// TIA Portal project "Bottle_line" (V15.1)

(* hardware
DEVICE "S7-1200 station_1"  S7-1200 Station
   slot 0: "Rack_0"  S7-1200 Rack  Rack  V1.0
   slot 1: "PLC_1"  CPU 1214C AC/DC/Rly  6ES7 214-1BG40-0XB0  V4.2
*)

// ===== PLC "PLC_1"  CPU 1214C AC/DC/Rly =====

VAR_GLOBAL   // PLC tag table "Default tag table"
   "System_Byte" AT %MB1 : Byte;
   "FirstScan" AT %M1.0 : Bool;
   "DiagStatusUpdate" AT %M1.1 : Bool;
   "AlwaysTRUE" AT %M1.2 : Bool;
   "AlwaysFALSE" AT %M1.3 : Bool;
   "Clock_Byte" AT %MB0 : Byte;
   "Clock_10Hz" AT %M0.0 : Bool;
   "Clock_5Hz" AT %M0.1 : Bool;
   "Clock_2.5Hz" AT %M0.2 : Bool;
   "Clock_2Hz" AT %M0.3 : Bool;
   "Clock_1.25Hz" AT %M0.4 : Bool;
   "Clock_1Hz" AT %M0.5 : Bool;
   "Clock_0.625Hz" AT %M0.6 : Bool;
   "Clock_0.5Hz" AT %M0.7 : Bool;
   "System_Byte(1)" AT %MB1 : Byte;
END_VAR

VAR_GLOBAL   // PLC tag table "Tag table_1"
   "LevelSensor" AT %IW56 : Word;
   "FlowMeter" AT %IW58 : Word;
   "FillTankValve" AT %QW56 : Word;
   "DrainValve" AT %QW58 : Word;
   "Start" AT %I20.0 : Bool;
   "Stop" AT %I20.1 : Bool;
   "Pause" AT %I20.2 : Bool;
   "BottleDetector" AT %I20.3 : Bool;
   "BottleCounter" AT %I20.4 : Bool;
   "BottleDetect" AT %I20.5 : Bool;
   "Emitter" AT %Q20.0 : Bool;
   "Conveyor1" AT %Q20.1 : Bool;
   "Conveyor2" AT %Q20.2 : Bool;
   "Conveyor3" AT %Q20.3 : Bool;
   "Conveyor4" AT %Q20.4 : Bool;
   "Conveyor5" AT %Q20.5 : Bool;
   "RollerStop" AT %Q20.6 : Bool;
   "RoboticArmZ" AT %Q20.7 : Bool;
   "GrabArmZ" AT %Q21.0 : Bool;
   "FillingLED" AT %Q21.1 : Bool;
   "GreenLED" AT %Q21.2 : Bool;
   "RedLEd" AT %Q21.3 : Bool;
   "YellowLED" AT %Q21.4 : Bool;
   "CounterDisplay" AT %QW60 : Word;
END_VAR

DATA_BLOCK "Bottle_Filling_DB"   // DB1
{ S7_Optimized_Access := 'TRUE' }
VERSION : 0.1
// stored: InstanceOfName Bottle_Filling
"Bottle_Filling"
BEGIN
END_DATA_BLOCK

DATA_BLOCK "Data"   // DB3
{ S7_Optimized_Access := 'TRUE' }
VERSION : 0.1
   VAR
      "SPTank(mm)" : Int := 3000;
      "PVTank(mm)" : Real;
      EnablePID : Bool;
      Norm : Real;
      "Caudal(m3/s)" : Real;
      bottleReset : Bool;
      "PVBottle(L)" : Real;
      "SPBottle(L)" : Real;
      BottleFill : Bool;
   END_VAR
BEGIN
END_DATA_BLOCK

DATA_BLOCK "Integration_DB"   // DB4
{ S7_Optimized_Access := 'TRUE' }
VERSION : 0.1
// stored: InstanceOfName Integration
"Integration"
BEGIN
END_DATA_BLOCK

DATA_BLOCK "TON_DB"   // DB7
{ S7_Optimized_Access := 'TRUE' }
VERSION : 0.1
// stored: InstanceOfName TON
"TON"
BEGIN
END_DATA_BLOCK

// folder: System blocks/Program resources

DATA_BLOCK "IEC_Timer_0_DB"   // DB6
{ S7_Optimized_Access := 'TRUE' }
AUTHOR : Simatic
FAMILY : IEC
NAME : IEC_TMR
VERSION : 1.0
// stored: InstanceOfName IEC_TIMER
"IEC_TIMER"
BEGIN
END_DATA_BLOCK

// folder: (top level)

FUNCTION_BLOCK "Bottle_Filling"   // FB1, LAD
{ S7_Optimized_Access := 'TRUE' }
VERSION : 0.1
   VAR_INPUT
      Start : Bool;
      Stop : Bool;
      Pause : Bool;
      BottleDetect : Bool;
      BottleCounter : Bool;
      BottleDetecter : Bool;
      LevelSensor : Int;
      "PV Bottle" : Real;
      "SP Bottle" : Real;
   END_VAR
   VAR_OUTPUT
      Emitter : Bool;
      Conveyor1 : Bool;
      Conveyor2 : Bool;
      Conveyor3 : Bool;
      Conveyor4 : Bool;
      Conveyor5 : Bool;
      RollerStop : Bool;
      RobotArmZ : Bool;
      GrabArmZ : Bool;
      FillingLED : Bool;
      GreenLED : Bool;
      RedLED : Bool;
      YellowLED : Bool;
      CounterDisplay : Int;
      LevelTank : Real;
      "BottleFilling X" : Bool;
      "BottleReset X" : Bool;
   END_VAR
   VAR
      K : Bool;
      Aux1 : Bool;
      Aux2 : Bool;
      X1_Emitter : Bool;
      X2_Emitter : Bool;
      Flanco1 : Bool;
      Flanco2 : Bool;
      Flanco3 : Bool;
      Flanco4 : Bool;
      XF : Bool;
      X1Stop : Bool;
      X2Stop : Bool;
      Detener : Bool;
      Norm : Real;
      "SP-error" : Real;
      "SP+error" : Real;
      "Counter" : CTU_INT;
      TON1 : "TON";
      TON3 : "TON";
      TON2 : "TON";
   END_VAR
   VAR_TEMP   // added for the SCL form of the ladder/FBD networks
      _w1 : Bool;
      _w2 : Bool;
   END_VAR
BEGIN

REGION Network 1
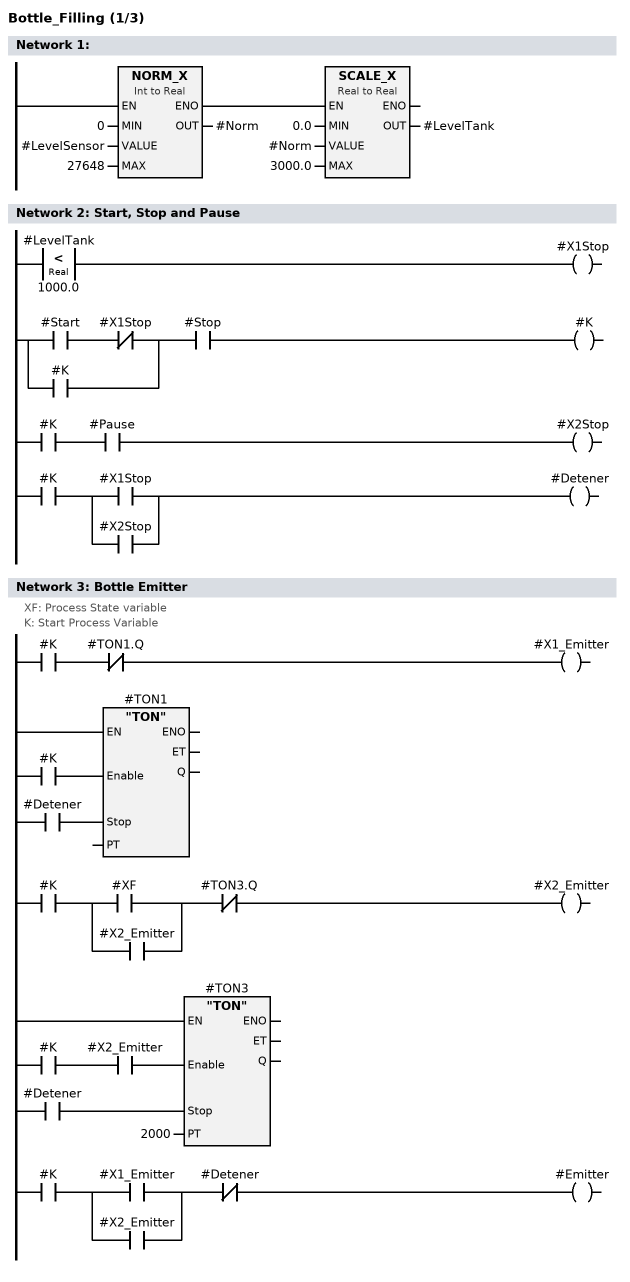
   RUNG wire#powerrail
      { S7_Templates := "[SrcType := Int, DestType := Real]" } Normalize(min := 0, value := #LevelSensor, max := 27648, out => #Norm)
      { S7_Templates := "[SrcType := Real, DestType := Real]" } Scale(min := 0.0, value := #Norm, max := 3000.0, out => #LevelTank)
   END_RUNG
   // the same network as SCL:
   #Norm := NORM_X(MIN := 0, VALUE := #LevelSensor, MAX := 27648);
   #LevelTank := SCALE_X(MIN := 0.0, VALUE := #Norm, MAX := 3000.0);
END_REGION

REGION Network 2: Start, Stop and Pause
   RUNG wire#powerrail
      { S7_Templates := "SrcType := Real" } LT_Contact(in1 := #LevelTank, in2 := 1000.0)
      Coil( #X1Stop )
   END_RUNG
   RUNG wire#powerrail
      Contact( #Start )
      I_Contact( #X1Stop )
      wire#w1
      Contact( #Stop )
      Coil( #K )
   END_RUNG
   RUNG wire#powerrail
      Contact( #K )
   END_RUNG wire#w1
   RUNG wire#powerrail
      Contact( #K )
      Contact( #Pause )
      Coil( #X2Stop )
   END_RUNG
   RUNG wire#powerrail
      Contact( #K )
      wire#w2
      Contact( #X1Stop )
      wire#w3
      Coil( #Detener )
   END_RUNG
   RUNG wire#w2
      Contact( #X2Stop )
   END_RUNG wire#w3
   // the same network as SCL:
   #X1Stop := #LevelTank < 1000.0;
   #K := ((#Start AND NOT #X1Stop) OR #K) AND #Stop;
   #X2Stop := #K AND #Pause;
   #Detener := #K AND (#X1Stop OR #X2Stop);
END_REGION

REGION Network 3: Bottle Emitter
   // XF: Process State variable
   // K: Start Process Variable
   RUNG wire#powerrail
      Contact( #K )
      I_Contact( #TON1.Q )
      Coil( #X1_Emitter )
   END_RUNG
   RUNG wire#powerrail
      #TON1(Enable := wire#w1, Stop := wire#w2, PT :=, ET =>, Q =>)
   END_RUNG
   RUNG wire#powerrail
      Contact( #K )
   END_RUNG wire#w1
   RUNG wire#powerrail
      Contact( #Detener )
   END_RUNG wire#w2
   RUNG wire#powerrail
      Contact( #K )
      wire#w3
      Contact( #XF )
      wire#w4
      I_Contact( #TON3.Q )
      Coil( #X2_Emitter )
   END_RUNG
   RUNG wire#w3
      Contact( #X2_Emitter )
   END_RUNG wire#w4
   RUNG wire#powerrail
      #TON3(Enable := wire#w5, Stop := wire#w6, PT := 2000, ET =>, Q =>)
   END_RUNG
   RUNG wire#powerrail
      Contact( #K )
      Contact( #X2_Emitter )
   END_RUNG wire#w5
   RUNG wire#powerrail
      Contact( #Detener )
   END_RUNG wire#w6
   RUNG wire#powerrail
      Contact( #K )
      wire#w7
      Contact( #X1_Emitter )
      wire#w8
      I_Contact( #Detener )
      Coil( #Emitter )
   END_RUNG
   RUNG wire#w7
      Contact( #X2_Emitter )
   END_RUNG wire#w8
   // the same network as SCL:
   #X1_Emitter := #K AND NOT #TON1.Q;
   #TON1(Enable := #K, Stop := #Detener);   // "TON"
   #X2_Emitter := #K AND (#XF OR #X2_Emitter) AND NOT #TON3.Q;
   #TON3(Enable := #K AND #X2_Emitter, Stop := #Detener, PT := 2000);   // "TON"
   #Emitter := #K AND (#X1_Emitter OR #X2_Emitter) AND NOT #Detener;
END_REGION

REGION Network 4: Process
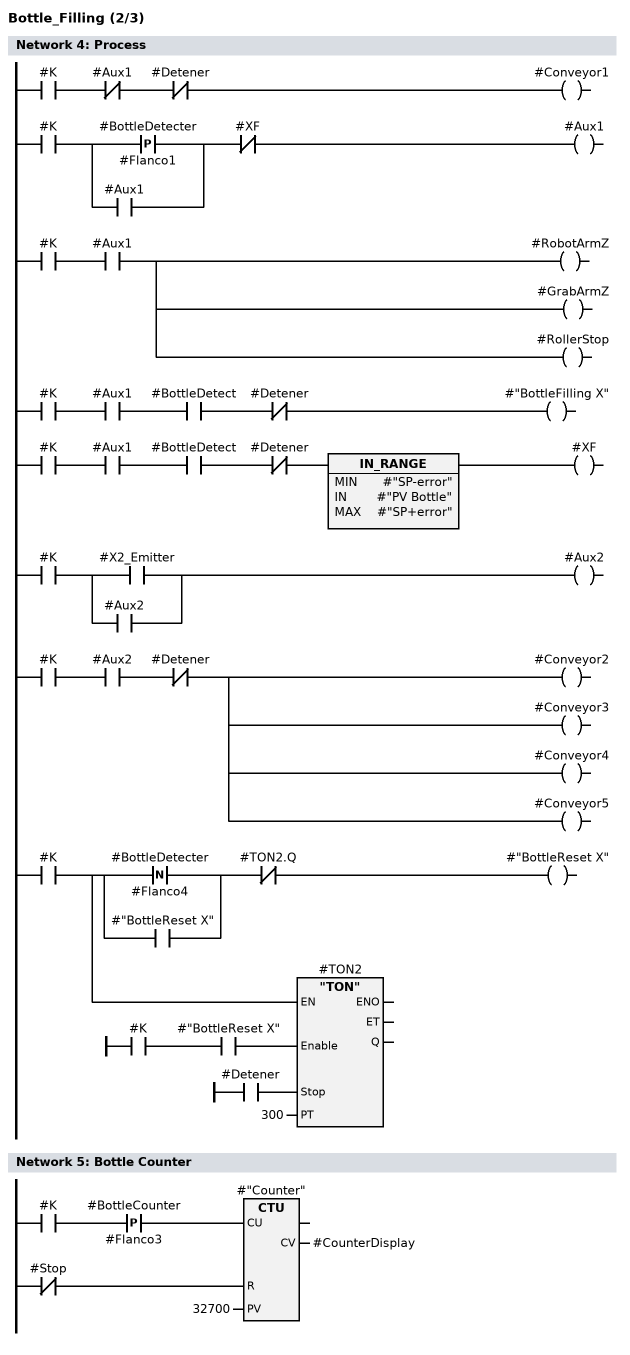
   RUNG wire#powerrail
      Contact( #K )
      I_Contact( #Aux1 )
      I_Contact( #Detener )
      Coil( #Conveyor1 )
   END_RUNG
   RUNG wire#powerrail
      Contact( #K )
      wire#w1
      P_Contact(operand := #BottleDetecter, bit := #Flanco1)
      wire#w2
      I_Contact( #XF )
      Coil( #Aux1 )
   END_RUNG
   RUNG wire#w1
      Contact( #Aux1 )
   END_RUNG wire#w2
   RUNG wire#powerrail
      Contact( #K )
      Contact( #Aux1 )
      wire#w3
      Coil( #RobotArmZ )
   END_RUNG
   RUNG wire#w3
      Coil( #GrabArmZ )
   END_RUNG
   RUNG wire#w3
      Coil( #RollerStop )
   END_RUNG
   RUNG wire#powerrail
      Contact( #K )
      Contact( #Aux1 )
      Contact( #BottleDetect )
      I_Contact( #Detener )
      Coil( #"BottleFilling X" )
   END_RUNG
   RUNG wire#powerrail
      Contact( #K )
      Contact( #Aux1 )
      Contact( #BottleDetect )
      I_Contact( #Detener )
      { S7_Templates := "SrcType := Real" } InRange(min := #"SP-error", in := #"PV Bottle", max := #"SP+error")
      Coil( #XF )
   END_RUNG
   RUNG wire#powerrail
      Contact( #K )
      wire#w4
      Contact( #X2_Emitter )
      wire#w5
      Coil( #Aux2 )
   END_RUNG
   RUNG wire#w4
      Contact( #Aux2 )
   END_RUNG wire#w5
   RUNG wire#powerrail
      Contact( #K )
      Contact( #Aux2 )
      I_Contact( #Detener )
      wire#w6
      Coil( #Conveyor2 )
   END_RUNG
   RUNG wire#w6
      Coil( #Conveyor3 )
   END_RUNG
   RUNG wire#w6
      Coil( #Conveyor4 )
   END_RUNG
   RUNG wire#w6
      Coil( #Conveyor5 )
   END_RUNG
   RUNG wire#powerrail
      Contact( #K )
      wire#w7
      N_Contact(operand := #BottleDetecter, bit := #Flanco4)
      wire#w8
      I_Contact( #TON2.Q )
      Coil( #"BottleReset X" )
   END_RUNG
   RUNG wire#w7
      Contact( #"BottleReset X" )
   END_RUNG wire#w8
   RUNG wire#w7
      #TON2(Enable := wire#w9, Stop := wire#w10, PT := 300, ET =>, Q =>)
   END_RUNG
   RUNG wire#powerrail
      Contact( #K )
      Contact( #"BottleReset X" )
   END_RUNG wire#w9
   RUNG wire#powerrail
      Contact( #Detener )
   END_RUNG wire#w10
   // the same network as SCL:
   #Conveyor1 := #K AND NOT #Aux1 AND NOT #Detener;
   #_w1 := #K AND #BottleDetecter AND NOT #Flanco1;   // rising edge of #BottleDetecter
   #Flanco1 := #BottleDetecter;
   #Aux1 := (#_w1 OR (#K AND #Aux1)) AND NOT #XF;
   #RobotArmZ := #K AND #Aux1;
   #GrabArmZ := #RobotArmZ;
   #RollerStop := #RobotArmZ;
   #"BottleFilling X" := #K AND #Aux1 AND #BottleDetect AND NOT #Detener;
   #XF := #K AND #Aux1 AND #BottleDetect AND NOT #Detener AND (#"SP-error" <= #"PV Bottle") AND (#"PV Bottle" <= #"SP+error");
   #Aux2 := #K AND (#X2_Emitter OR #Aux2);
   #Conveyor2 := #K AND #Aux2 AND NOT #Detener;
   #Conveyor3 := #Conveyor2;
   #Conveyor4 := #Conveyor2;
   #Conveyor5 := #Conveyor2;
   #_w2 := #K AND NOT #BottleDetecter AND #Flanco4;   // falling edge of #BottleDetecter
   #Flanco4 := #BottleDetecter;
   #"BottleReset X" := (#_w2 OR (#K AND #"BottleReset X")) AND NOT #TON2.Q;
   IF #K THEN
       #TON2(Enable := #K AND #"BottleReset X", Stop := #Detener, PT := 300);   // "TON"
   END_IF;
END_REGION

REGION Network 5: Bottle Counter
   #_w1 := #K AND #BottleCounter AND NOT #Flanco3;   // rising edge of #BottleCounter
   #Flanco3 := #BottleCounter;
   #"Counter"(CU := #_w1, R := NOT #Stop, PV := 32700, CV => #CounterDisplay);   // CTU
END_REGION

REGION Network 6: Light Control
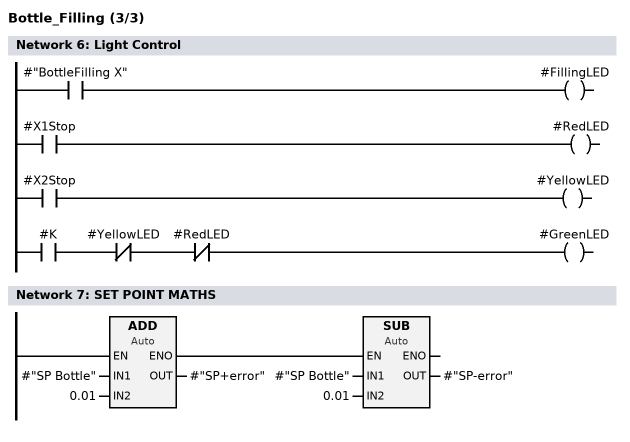
   RUNG wire#powerrail
      Contact( #"BottleFilling X" )
      Coil( #FillingLED )
   END_RUNG
   RUNG wire#powerrail
      Contact( #X1Stop )
      Coil( #RedLED )
   END_RUNG
   RUNG wire#powerrail
      Contact( #X2Stop )
      Coil( #YellowLED )
   END_RUNG
   RUNG wire#powerrail
      Contact( #K )
      I_Contact( #YellowLED )
      I_Contact( #RedLED )
      Coil( #GreenLED )
   END_RUNG
   // the same network as SCL:
   #FillingLED := #"BottleFilling X";
   #RedLED := #X1Stop;
   #YellowLED := #X2Stop;
   #GreenLED := #K AND NOT #YellowLED AND NOT #RedLED;
END_REGION

REGION Network 7: SET POINT MATHS
   RUNG wire#powerrail
      Add(in1 := #"SP Bottle", in2 := 0.01, out => #"SP+error")
      Sub(in1 := #"SP Bottle", in2 := 0.01, out => #"SP-error")
   END_RUNG
   // the same network as SCL:
   #"SP+error" := #"SP Bottle" + 0.01;
   #"SP-error" := #"SP Bottle" - 0.01;
END_REGION
END_FUNCTION_BLOCK

FUNCTION_BLOCK "TON"   // FB2, LAD
{ S7_Optimized_Access := 'TRUE' }
VERSION : 0.1
   VAR_INPUT
      Enable : Bool;
      Stop : Bool;
      PT : Int;
   END_VAR
   VAR_OUTPUT
      ET : Int;
      Q : Bool;
   END_VAR
   VAR_TEMP
      TimeAux : Time;
      ETAux : Time;
   END_VAR
BEGIN

REGION Network 1
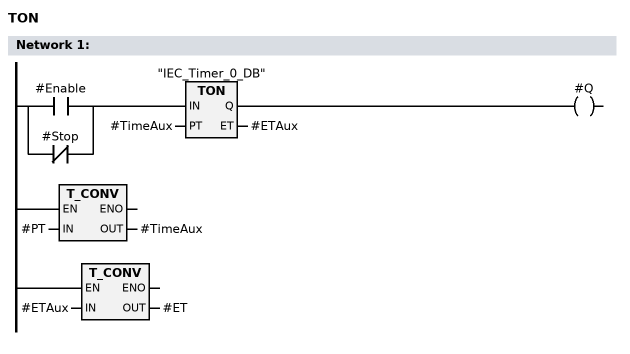
   "IEC_Timer_0_DB".TON(IN := #Enable OR NOT #Stop, PT := #TimeAux, ET => #ETAux);
   #Q := "IEC_Timer_0_DB".Q;
   #TimeAux := T_CONV(IN := #PT);
   #ET := T_CONV(IN := #ETAux);
END_REGION
END_FUNCTION_BLOCK

FUNCTION_BLOCK "Analogic"   // FB3, LAD
{ S7_Optimized_Access := 'TRUE' }
VERSION : 0.1
BEGIN
END_FUNCTION_BLOCK

FUNCTION_BLOCK "Integration"   // FB4, LAD
{ S7_Optimized_Access := 'TRUE' }
VERSION : 0.1
   VAR_INPUT
      Enable : Bool;
      "Tm(ms)" : Real;
      Signal : Real;
      SignalFormat : Real;
      Reset : Bool;
   END_VAR
   VAR_OUTPUT
      Integral : Real;
   END_VAR
   VAR_TEMP
      DeltaVol : Real;
      VolTotal : Real;
      FormatedSignal : Real;
      DeltaTime : Real;
      Result_2 : Real;
   END_VAR
BEGIN

REGION Network 1
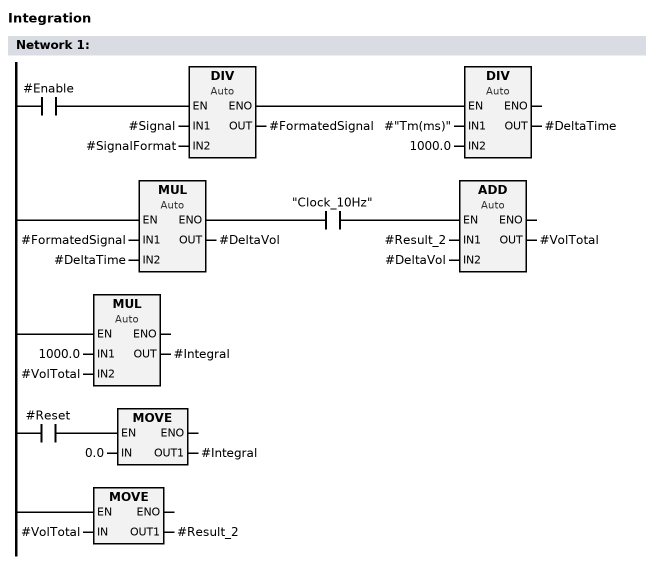
   RUNG wire#powerrail
      Contact( #Enable )
      Div(in1 := #Signal, in2 := #SignalFormat, out => #FormatedSignal)
      Div(in1 := #"Tm(ms)", in2 := 1000.0, out => #DeltaTime)
   END_RUNG
   RUNG wire#powerrail
      Mul(in1 := #FormatedSignal, in2 := #DeltaTime, out => #DeltaVol)
      Contact( "Clock_10Hz" )
      Add(in1 := #Result_2, in2 := #DeltaVol, out => #VolTotal)
   END_RUNG
   RUNG wire#powerrail
      Mul(in1 := 1000.0, in2 := #VolTotal, out => #Integral)
   END_RUNG
   RUNG wire#powerrail
      Contact( #Reset )
      Move(in := 0.0, out1 => #Integral)
   END_RUNG
   RUNG wire#powerrail
      Move(in := #VolTotal, out1 => #Result_2)
   END_RUNG
   // the same network as SCL:
   IF #Enable THEN
       #FormatedSignal := #Signal / #SignalFormat;
       #DeltaTime := #"Tm(ms)" / 1000.0;
   END_IF;
   #DeltaVol := #FormatedSignal * #DeltaTime;
   IF "Clock_10Hz" THEN #VolTotal := #Result_2 + #DeltaVol; END_IF;
   #Integral := 1000.0 * #VolTotal;
   IF #Reset THEN #Integral := 0.0; END_IF;
   #Result_2 := #VolTotal;
END_REGION
END_FUNCTION_BLOCK

FUNCTION "MHJ-PLC-Lab-Function-S71200" : Void   // FC1, SCL
{ S7_Optimized_Access := 'TRUE' }
VERSION : 0.1
   VAR_TEMP
      rdTimeReturn : Int;
      outputTime : DTL;
      SyncVal : Byte;
      forVal : Int;
      forVal_2 : Int;
      Value : Byte;
   END_VAR
   VAR CONSTANT
      CompVal : Byte := 16#34;
      Value_01 : Byte := 16#11;
      Value_01_DW : DWord := 16#A165_D992;
      Value_02_DW : DWord := 16#58BE_4401;
   END_VAR
BEGIN

   #Value := PEEK(area := 16#82,
                  dbNumber := 0,
                  byteOffset := 511);
   #Value := #Value + 1;

   POKE(area := 16#82,
        dbNumber := 0,
        byteOffset := 511,
        value := #Value);

   POKE(area := 16#81,
        dbNumber := 0,
        byteOffset := 1016,
        value := #Value_01_DW);
   POKE(area := 16#81,
        dbNumber := 0,
        byteOffset := 1020,
        value := #Value_02_DW);

   POKE(area := 16#81,
        dbNumber := 0,
        byteOffset := 511,
        value := B#16#00);

   FOR #forVal := 0 TO 120 DO
       FOR #forVal_2 := 0 TO 10 DO
           #rdTimeReturn := RD_SYS_T(#outputTime);
           #rdTimeReturn := WR_SYS_T(#outputTime);
           #rdTimeReturn := RD_SYS_T(#outputTime);
           #rdTimeReturn := WR_SYS_T(#outputTime);
       END_FOR;
       #SyncVal := PEEK(area := 16#81,
                        dbNumber := 0,
                        byteOffset := 511);
       IF #SyncVal = #CompVal THEN
           GOTO M_1;
       END_IF;
   END_FOR;
   RETURN;

   M_1:
   POKE(area := 16#81,
        dbNumber := 0,
        byteOffset := 511,
        value := B#16#0);
END_FUNCTION

ORGANIZATION_BLOCK "Main"   // OB1, LAD, ProgramCycle
TITLE = "Main Program Sweep (Cycle)"
{ S7_Optimized_Access := 'TRUE' }
VERSION : 0.1
   VAR_INPUT
      Initial_Call : Bool;   // Initial call of this OB
      Remanence : Bool;   // =True, if remanent data are available
   END_VAR
BEGIN

REGION Network 1
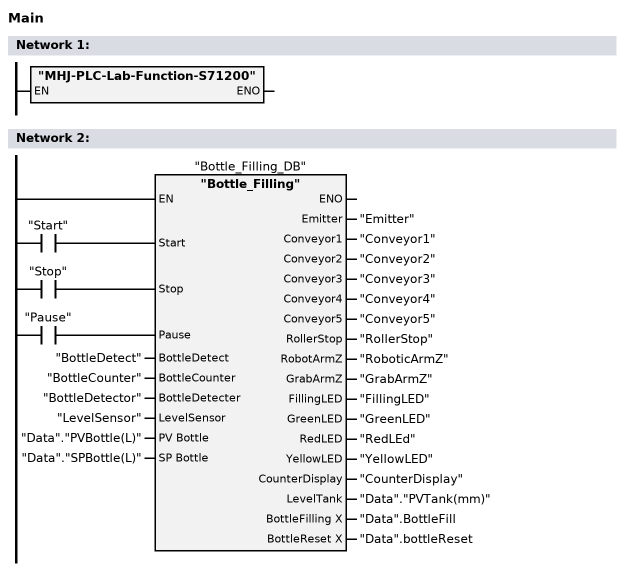
   RUNG wire#powerrail
      "MHJ-PLC-Lab-Function-S71200"()
   END_RUNG
   // the same network as SCL:
   "MHJ-PLC-Lab-Function-S71200"();
END_REGION

REGION Network 2
   RUNG wire#powerrail
      "Bottle_Filling_DB"(Start := wire#w1, Stop := wire#w2, Pause := wire#w3, BottleDetect := "BottleDetect", BottleCounter := "BottleCounter", BottleDetecter := "BottleDetector", LevelSensor := "LevelSensor", "PV Bottle" := "Data"."PVBottle(L)", "SP Bottle" := "Data"."SPBottle(L)", Emitter => "Emitter", Conveyor1 => "Conveyor1", Conveyor2 => "Conveyor2", Conveyor3 => "Conveyor3", Conveyor4 => "Conveyor4", Conveyor5 => "Conveyor5", RollerStop => "RollerStop", RobotArmZ => "RoboticArmZ", GrabArmZ => "GrabArmZ", FillingLED => "FillingLED", GreenLED => "GreenLED", RedLED => "RedLEd", YellowLED => "YellowLED", CounterDisplay => "CounterDisplay", LevelTank => "Data"."PVTank(mm)", "BottleFilling X" => "Data".BottleFill, "BottleReset X" => "Data".bottleReset)
   END_RUNG
   RUNG wire#powerrail
      Contact( "Start" )
   END_RUNG wire#w1
   RUNG wire#powerrail
      Contact( "Stop" )
   END_RUNG wire#w2
   RUNG wire#powerrail
      Contact( "Pause" )
   END_RUNG wire#w3
   // the same network as SCL:
   "Bottle_Filling_DB"(Start := "Start",   // "Bottle_Filling"
                       Stop := "Stop",
                       Pause := "Pause",
                       BottleDetect := "BottleDetect",
                       BottleCounter := "BottleCounter",
                       BottleDetecter := "BottleDetector",
                       LevelSensor := "LevelSensor",
                       "PV Bottle" := "Data"."PVBottle(L)",
                       "SP Bottle" := "Data"."SPBottle(L)",
                       Emitter => "Emitter",
                       Conveyor1 => "Conveyor1",
                       Conveyor2 => "Conveyor2",
                       Conveyor3 => "Conveyor3",
                       Conveyor4 => "Conveyor4",
                       Conveyor5 => "Conveyor5",
                       RollerStop => "RollerStop",
                       RobotArmZ => "RoboticArmZ",
                       GrabArmZ => "GrabArmZ",
                       FillingLED => "FillingLED",
                       GreenLED => "GreenLED",
                       RedLED => "RedLEd",
                       YellowLED => "YellowLED",
                       CounterDisplay => "CounterDisplay",
                       LevelTank => "Data"."PVTank(mm)",
                       "BottleFilling X" => "Data".BottleFill,
                       "BottleReset X" => "Data".bottleReset);
END_REGION
END_ORGANIZATION_BLOCK

ORGANIZATION_BLOCK "Cyclic interrupt"   // OB30, LAD, CyclicInterrupt
{ S7_Optimized_Access := 'TRUE' }
VERSION : 0.1
   VAR_INPUT
      Initial_Call : Bool;   // Initial call of this OB
      Event_Count : Int;   // Events discarded
   END_VAR
BEGIN

REGION Network 1: PID Level Tank Control
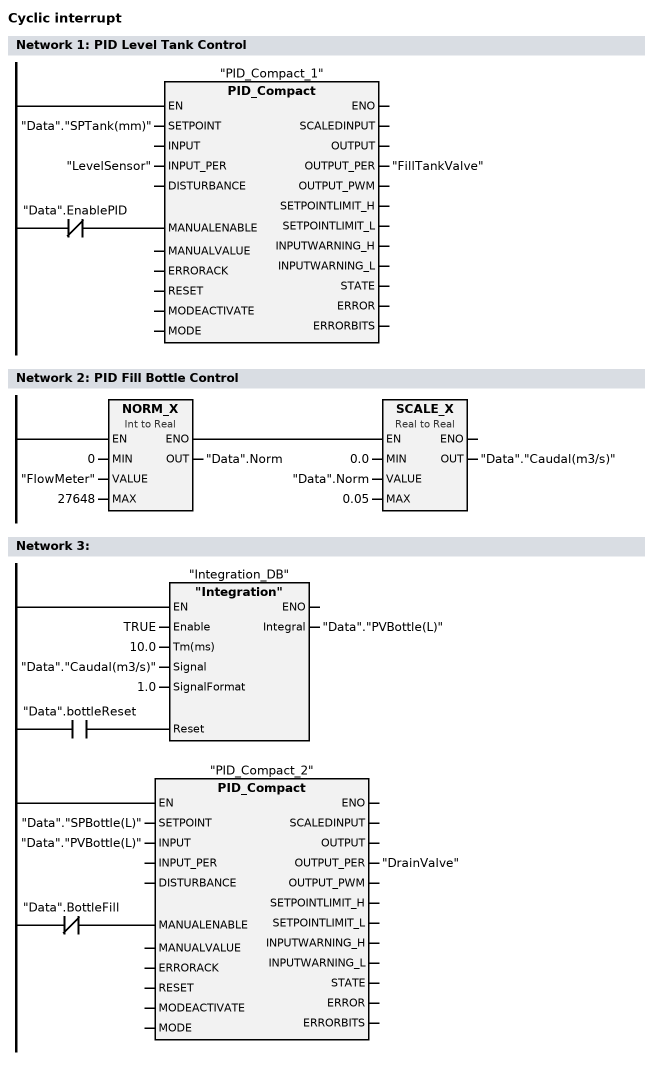
   "PID_Compact_1"(Setpoint := "Data"."SPTank(mm)",   // PID_Compact
                   Input_PER := "LevelSensor",
                   ManualEnable := NOT "Data".EnablePID,
                   Output_PER => "FillTankValve");
END_REGION

REGION Network 2: PID Fill Bottle Control
   RUNG wire#powerrail
      { S7_Templates := "[SrcType := Int, DestType := Real]" } Normalize(min := 0, value := "FlowMeter", max := 27648, out => "Data".Norm)
      { S7_Templates := "[SrcType := Real, DestType := Real]" } Scale(min := 0.0, value := "Data".Norm, max := 0.05, out => "Data"."Caudal(m3/s)")
   END_RUNG
   // the same network as SCL:
   "Data".Norm := NORM_X(MIN := 0, VALUE := "FlowMeter", MAX := 27648);
   "Data"."Caudal(m3/s)" := SCALE_X(MIN := 0.0, VALUE := "Data".Norm, MAX := 0.05);
END_REGION

REGION Network 3
   "Integration_DB"(Enable := TRUE,   // "Integration"
                    "Tm(ms)" := 10.0,
                    Signal := "Data"."Caudal(m3/s)",
                    SignalFormat := 1.0,
                    Reset := "Data".bottleReset,
                    Integral => "Data"."PVBottle(L)");
   "PID_Compact_2"(Setpoint := "Data"."SPBottle(L)",   // PID_Compact
                   Input := "Data"."PVBottle(L)",
                   ManualEnable := NOT "Data".BottleFill,
                   Output_PER => "DrainValve");
END_REGION
END_ORGANIZATION_BLOCK